Yaskawa INFORM job: AAA.JBI

/JOB
//NAME AAA
//POS
///NPOS 102,0,0,0,0,0
///TOOL 11
///POSTYPE PULSE
///PULSE
C00000=-47590,-794,-17593,-13589,-96385,55915
C00001=-47590,-794,-17593,-13589,-96385,55915
C00002=-44371,-5320,-21356,-14077,-96305,55735
C00003=-43831,-6151,-22025,-14192,-96253,55715
C00004=-43310,-7063,-22747,-14335,-96160,55710
C00005=-42810,-8059,-23521,-14506,-96026,55720
C00006=-42328,-9139,-24348,-14702,-95852,55745
C00007=-41866,-10304,-25228,-14925,-95638,55784
C00008=-41422,-11555,-26161,-15172,-95384,55837
C00009=-40996,-12894,-27148,-15444,-95090,55904
C00010=-40589,-14321,-28187,-15740,-94756,55986
C00011=-40200,-15836,-29280,-16060,-94383,56080
C00012=-39827,-17440,-30427,-16403,-93972,56188
C00013=-39472,-19134,-31627,-16768,-93524,56309
C00014=-39134,-20916,-32880,-17155,-93040,56442
C00015=-38811,-22786,-34184,-17564,-92521,56585
C00016=-38503,-24741,-35540,-17994,-91968,56739
C00017=-38210,-26781,-36944,-18445,-91384,56902
C00018=-37930,-28901,-38396,-18915,-90772,57072
C00019=-37661,-31098,-39892,-19404,-90132,57248
C00020=-37403,-33367,-41430,-19911,-89470,57427
C00021=-37153,-35704,-43004,-20434,-88786,57608
C00022=-36909,-38100,-44611,-20972,-88086,57787
C00023=-36669,-40550,-46246,-21523,-87371,57961
C00024=-36429,-43044,-47903,-22085,-86647,58127
C00025=-36188,-45575,-49575,-22655,-85916,58280
C00026=-35942,-48131,-51256,-23232,-85182,58416
C00027=-35687,-50704,-52938,-23812,-84448,58531
C00028=-35420,-53282,-54614,-24392,-83718,58619
C00029=-35137,-55853,-56275,-24969,-82995,58675
C00030=-34833,-58405,-57914,-25540,-82281,58693
C00031=-34505,-60927,-59521,-26100,-81578,58667
C00032=-34148,-63405,-61088,-26646,-80889,58591
C00033=-33757,-65825,-62605,-27172,-80214,58458
C00034=-33329,-68174,-64064,-27675,-79555,58263
C00035=-32857,-70435,-65454,-28149,-78913,57999
C00036=-32337,-72593,-66764,-28588,-78288,57660
C00037=-31763,-74629,-67984,-28985,-77682,57242
C00038=-31130,-76523,-69101,-29332,-77095,56739
C00039=-30431,-78252,-70100,-29621,-76530,56149
C00040=-29662,-79790,-70968,-29842,-75989,55468
C00041=-28816,-81106,-71686,-29985,-75477,54697
C00042=-27889,-82170,-72236,-30040,-74999,53835
C00043=-26877,-82945,-72599,-29996,-74565,52886
C00044=-25776,-83390,-72752,-29844,-74187,51855
C00045=-24589,-83462,-72672,-29579,-73879,50748
C00046=-23317,-83120,-72338,-29195,-73661,49577
C00047=-21969,-82322,-71728,-28696,-73553,48352
C00048=-20555,-81028,-70822,-28088,-73579,47088
C00049=-19089,-79207,-69607,-27384,-73766,45797
C00050=-17588,-76837,-68070,-26604,-74137,44495
C00051=-16073,-73906,-66210,-25772,-74715,43196
C00052=-14563,-70418,-64032,-24916,-75518,41915
C00053=-13081,-66394,-61550,-24067,-76558,40664
C00054=-11644,-61874,-58793,-23255,-77836,39457
C00055=-10271,-56916,-55800,-22510,-79344,38302
C00056=-8973,-51601,-52622,-21856,-81060,37211
C00057=-7761,-46025,-49323,-21312,-82953,36192
C00058=-6639,-40297,-45973,-20891,-84980,35254
C00059=-5608,-34529,-42643,-20599,-87094,34408
C00060=-4665,-28836,-39403,-20439,-89243,33667
C00061=-3804,-23313,-36312,-20406,-91382,33044
C00062=-3018,-18045,-33417,-20495,-93471,32556
C00063=-2299,-13094,-30751,-20698,-95478,32222
C00064=-1638,-8506,-28332,-21004,-97382,32063
C00065=-1026,-4306,-26170,-21403,-99172,32100
C00066=-453,-510,-24261,-21881,-100843,32352
C00067=93,2872,-22599,-22421,-102392,32835
C00068=626,5829,-21178,-22999,-103818,33558
C00069=1159,8338,-19993,-23587,-105109,34516
C00070=1709,10361,-19045,-24145,-106243,35686
C00071=2286,11842,-18345,-24634,-107181,37026
C00072=2903,12711,-17913,-25017,-107871,38476
C00073=3560,12885,-17780,-25267,-108249,39965
C00074=4257,12287,-17987,-25373,-108253,41425
C00075=4988,10851,-18575,-25338,-107831,42797
C00076=5751,8528,-19592,-25174,-106943,44045
C00077=6547,5286,-21081,-24900,-105570,45150
C00078=7382,1120,-23079,-24535,-103708,46106
C00079=8269,-3948,-25611,-24099,-101376,46915
C00080=9225,-9852,-28675,-23607,-98612,47582
C00081=10264,-16475,-32233,-23073,-95484,48105
C00082=11400,-23643,-36206,-22507,-92080,48476
C00083=12641,-31141,-40477,-21920,-88504,48675
C00084=13981,-38738,-44909,-21319,-84862,48674
C00085=15408,-46214,-49362,-20713,-81244,48431
C00086=16898,-53388,-53714,-20114,-77718,47903
C00087=18426,-60129,-57869,-19532,-74317,47034
C00088=19969,-66345,-61760,-18968,-71052,45765
C00089=21519,-71964,-65325,-18401,-67917,44036
C00090=23084,-76882,-68487,-17770,-64920,41795
C00091=24682,-80910,-71115,-16983,-62116,39041
C00092=26307,-83749,-73010,-15956,-59645,35864
C00093=27884,-85043,-73939,-14718,-57721,32478
C00094=29264,-84509,-73712,-13471,-56570,29191
C00095=30275,-82064,-72253,-12521,-56335,26293
C00096=30803,-77811,-69608,-12125,-57055,23962
C00097=30828,-71963,-65898,-12378,-58686,22231
C00098=30408,-64777,-61292,-13224,-61139,21030
C00099=29655,-56531,-55993,-14515,-64291,20234
C00100=28704,-47548,-50241,-16082,-67978,19722
C00101=23915,4176,-18337,-25769,-91161,16957
//INST
///DATE 2023/05/03 14:56
///ATTR SC,RW
///GROUP1 RB1
NOP
MOVJ C00000 VJ=5.0
TIMER T=1.00
MOVJ C00001 VJ=1.0
TIMER T=0.10
MOVL C00002 V=200.0 PL=8
MOVL C00003 V=200.0 PL=8
MOVL C00004 V=200.0 PL=8
MOVL C00005 V=200.0 PL=8
MOVL C00006 V=200.0 PL=8
MOVL C00007 V=200.0 PL=8
MOVL C00008 V=200.0 PL=8
MOVL C00009 V=200.0 PL=8
MOVL C00010 V=200.0 PL=8
MOVL C00011 V=200.0 PL=8
MOVL C00012 V=200.0 PL=8
MOVL C00013 V=200.0 PL=8
MOVL C00014 V=200.0 PL=8
MOVL C00015 V=200.0 PL=8
MOVL C00016 V=200.0 PL=8
MOVL C00017 V=200.0 PL=8
MOVL C00018 V=200.0 PL=8
MOVL C00019 V=200.0 PL=8
MOVL C00020 V=200.0 PL=8
MOVL C00021 V=200.0 PL=8
MOVL C00022 V=200.0 PL=8
MOVL C00023 V=200.0 PL=8
MOVL C00024 V=200.0 PL=8
MOVL C00025 V=200.0 PL=8
MOVL C00026 V=200.0 PL=8
MOVL C00027 V=200.0 PL=8
MOVL C00028 V=200.0 PL=8
MOVL C00029 V=200.0 PL=8
MOVL C00030 V=200.0 PL=8
MOVL C00031 V=200.0 PL=8
MOVL C00032 V=200.0 PL=8
MOVL C00033 V=200.0 PL=8
MOVL C00034 V=200.0 PL=8
MOVL C00035 V=200.0 PL=8
MOVL C00036 V=200.0 PL=8
MOVL C00037 V=200.0 PL=8
MOVL C00038 V=200.0 PL=8
MOVL C00039 V=200.0 PL=8
MOVL C00040 V=200.0 PL=8
MOVL C00041 V=200.0 PL=8
MOVL C00042 V=200.0 PL=8
MOVL C00043 V=200.0 PL=8
MOVL C00044 V=200.0 PL=8
MOVL C00045 V=200.0 PL=8
MOVL C00046 V=200.0 PL=8
MOVL C00047 V=200.0 PL=8
MOVL C00048 V=200.0 PL=8
MOVL C00049 V=200.0 PL=8
MOVL C00050 V=200.0 PL=8
MOVL C00051 V=200.0 PL=8
MOVL C00052 V=200.0 PL=8
MOVL C00053 V=200.0 PL=8
MOVL C00054 V=200.0 PL=8
MOVL C00055 V=200.0 PL=8
MOVL C00056 V=200.0 PL=8
MOVL C00057 V=200.0 PL=8
MOVL C00058 V=200.0 PL=8
MOVL C00059 V=200.0 PL=8
MOVL C00060 V=200.0 PL=8
MOVL C00061 V=200.0 PL=8
MOVL C00062 V=200.0 PL=8
MOVL C00063 V=200.0 PL=8
MOVL C00064 V=200.0 PL=8
MOVL C00065 V=200.0 PL=8
MOVL C00066 V=200.0 PL=8
MOVL C00067 V=200.0 PL=8
MOVL C00068 V=200.0 PL=8
MOVL C00069 V=200.0 PL=8
MOVL C00070 V=200.0 PL=8
MOVL C00071 V=200.0 PL=8
MOVL C00072 V=200.0 PL=8
MOVL C00073 V=200.0 PL=8
MOVL C00074 V=200.0 PL=8
MOVL C00075 V=200.0 PL=8
MOVL C00076 V=200.0 PL=8
MOVL C00077 V=200.0 PL=8
MOVL C00078 V=200.0 PL=8
MOVL C00079 V=200.0 PL=8
MOVL C00080 V=200.0 PL=8
MOVL C00081 V=200.0 PL=8
MOVL C00082 V=200.0 PL=8
MOVL C00083 V=200.0 PL=8
MOVL C00084 V=200.0 PL=8
MOVL C00085 V=200.0 PL=8
MOVL C00086 V=200.0 PL=8
MOVL C00087 V=200.0 PL=8
MOVL C00088 V=200.0 PL=8
MOVL C00089 V=200.0 PL=8
MOVL C00090 V=200.0 PL=8
MOVL C00091 V=200.0 PL=8
MOVL C00092 V=200.0 PL=8
MOVL C00093 V=200.0 PL=8
MOVL C00094 V=200.0 PL=8
MOVL C00095 V=200.0 PL=8
MOVL C00096 V=200.0 PL=8
MOVL C00097 V=200.0 PL=8
MOVL C00098 V=200.0 PL=8
MOVL C00099 V=200.0 PL=8
MOVL C00100 V=200.0 PL=8
MOVL C00101 V=200.0 PL=8
END
